// TIA Portal V17 export
BLOCK "FC_Timers"   // ObjectSW12, LAD
BEGIN

REGION Network 1: ton
END_REGION

REGION Network 2: tof
END_REGION

REGION Network 3: tp
END_REGION

REGION Network 4: tonr
END_REGION
END_BLOCK
